{region '#Template'}
	{attribute 'Category' := 'AC'}
	{attribute 'Version' := '0.0.1.0'}
	{attribute 'Tags' := 'AC, Aggregates, ERC, Temperature, Controller'}
	{attribute 'Description' := 'Energie Rückgewinnung Zuluft Regler Temperatur	// Energy recovery Supply air controller temperature'}
{endregion}
FUNCTION_BLOCK FB_BA_AC_ErcTSuACtrl EXTENDS FB_BA_View
VAR_INPUT
	bEn					: BOOL;
	fSpTSuA				: REAL;
	fTSuA				: REAL;
	bSync				: BOOL;
	fSync				: REAL;
	bDeHum				: BOOL;
	fTExtA				: REAL;
	fTWth				: REAL;
END_VAR
VAR_OUTPUT
	fY					: REAL;
	eAction				: E_BA_Action;
	bIsActive			: BOOL;	//	active sequence controller
	bOpState			: BOOL;	//	Release sequence link, sequence control is active	
END_VAR
VAR_INPUT CONSTANT PERSISTENT
	{attribute 'parameterCategory' := 'Behaviour'}
	fHysActionOn 		: REAL := 0.25;
	{attribute 'parameterCategory' := 'Behaviour'}
	fHysActionOff 		: REAL := -0.25;
END_VAR
VAR_INPUT CONSTANT
	Ctrl				: FB_BA_Loop;		 
END_VAR
VAR		
	HysAction			: FB_BA_Swi2P;
END_VAR

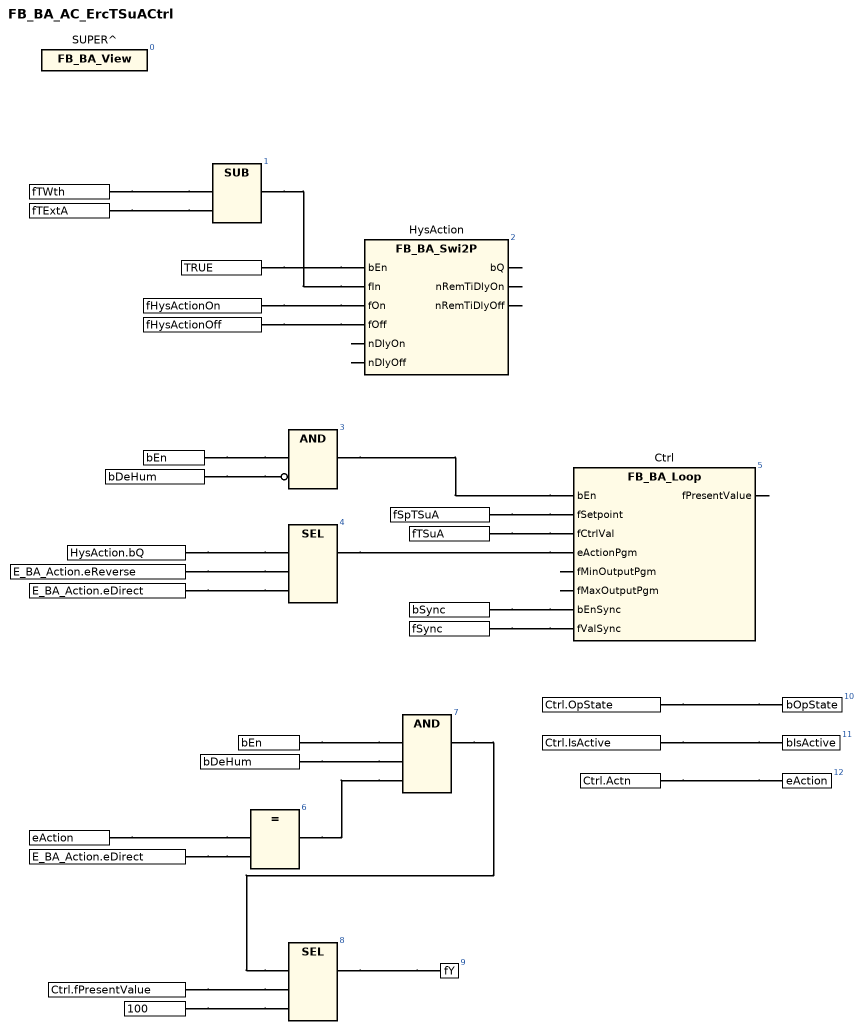
SUPER^(); // FB_BA_View
HysAction(bEn := TRUE, fIn := fTWth - fTExtA, fOn := fHysActionOn, fOff := fHysActionOff); // FB_BA_Swi2P
Ctrl(
    bEn := bEn AND NOT bDeHum,
    fSetpoint := fSpTSuA,
    fCtrlVal := fTSuA,
    eActionPgm := SEL(HysAction.bQ, E_BA_Action.eReverse, E_BA_Action.eDirect),
    bEnSync := bSync,
    fValSync := fSync); // FB_BA_Loop
fY := SEL(bEn AND bDeHum AND eAction = E_BA_Action.eDirect, Ctrl.fPresentValue, 100);
bOpState := Ctrl.OpState;
bIsActive := Ctrl.IsActive;
eAction := Ctrl.Actn;

METHOD FB_init : BOOL
VAR_INPUT
	bInitRetains : BOOL; // if TRUE, the retain variables are initialized (warm start / cold start)
	bInCopyCode : BOOL;  // if TRUE, the instance afterwards gets moved into the copy code (online change)
END_VAR
Ctrl.iParent						:= THIS^;
Ctrl.iLabel							:= LblCmpAC.ERC_TSuACtrl_Ctrl; 
Ctrl.sObjectName					:= '{Idx=01}';
Ctrl.eOpMode						:= BA2_Param.nLoop_DefOpMode;								 	 										 
Ctrl.eOutputUnit					:= E_BA_Unit.eOther_Percent;
Ctrl.eActionRm						:= E_BA_Action.eReverse;
Ctrl.fProportionalConstant			:= 3;
Ctrl.fIntegralConstant				:= 180;
Ctrl.fDerivativeConstant			:= 0;
Ctrl.fMaxOutputRm 					:= 100;
Ctrl.fMinOutputRm					:= 0;
Ctrl.fCOVIncrement					:= 0;
Ctrl.nDampConstant					:= 0;
Ctrl.fNeutralZone					:= 0;
Ctrl.stStepDelay.nDown				:= 0;
Ctrl.stStepDelay.nUp				:= 0;
END_METHOD

END_FUNCTION_BLOCK

(* stored: Version 1.1.0.1, ProductVersion 3.1.4024.6
   POU FB_BA_AC_ErcTSuACtrl: Id {87e72ae2-272a-4db0-8a4b-212d1ccec40e}, SpecialFunc None
   Method FB_init: Id {20981195-08fd-44f7-b2da-3335d736fc79} *)
